// TIA Portal V20 export
TYPE "typeEm2Parameter"
// stored: Namespace Unit1.Em2
   STRUCT
      "Bool" { ExternalAccessible := 'False'; ExternalVisible := 'False'; ExternalWritable := 'False'} : Array[0..50] of Bool;
      Data { ExternalAccessible := 'False'; ExternalVisible := 'False'; ExternalWritable := 'False'} : Array[0..50] of LReal;
   END_STRUCT;
END_TYPE
